{attribute addProperty BoxType "EL2521-0000-1022"}
{attribute addProperty Id "StatusAT %I*Status_9F9ED431162"}
{attribute addProperty CRC "657713736"}
{attribute addProperty SizeInBites "16"}
{attribute addProperty SizeInBytes "2"}
TYPE PTO_Status_2733EA48 :
STRUCT
	{attribute addProperty Name "Status"}
	Status AT %I* : Status_9F9ED431;
END_STRUCT
END_TYPE

(* stored: Version 1.2.0.0, ProductVersion 3.1.4024.9
   DUT PTO_Status_2733EA48: Id {0b33ad48-c305-4c8d-95f9-1ac9f50170ce} *)
